// TIA Portal V16 export
// export: Created 2024-03-28T09:48:21.6604235Z, ExportSetting WithDefaults, DisplayName Totally Integrated Automation Portal, DisplayVersion V16, DisplayName TIA Portal Version Control Interface, DisplayVersion V16, DisplayName TIA Portal Openness, DisplayVersion V16, DisplayName STEP 7 Professional, DisplayVersion V16, DisplayName STEP 7 Safety, DisplayVersion V16, DisplayName WinCC Advanced, DisplayVersion V16
TYPE "UR__T2O_Tool"
// stored: IsFailsafeCompliant false
   STRUCT
      "Tool mode" : USInt;
      Reserved_7_15 { ExternalAccessible := 'False'; ExternalVisible := 'False'; ExternalWritable := 'False'} : USInt;
      Reserved_16_31 { ExternalAccessible := 'False'; ExternalVisible := 'False'; ExternalWritable := 'False'} : UInt;
      "TDI: Tool Digital Inputs" : USInt;
      "TDO: Tool Digital Outputs" : USInt;
      "TAIT: Tool Analog Input Types" : USInt;
      Reserved_24_31 { ExternalAccessible := 'False'; ExternalVisible := 'False'; ExternalWritable := 'False'} : USInt;
      "Tool analog input [A or V]" : Array[0..1] of Real;
      "Tool output voltage [V]" : Real;
      "Tool current [A]" : Real;
   END_STRUCT;
END_TYPE
